TYPE ST_SortStationParam :
STRUCT
	lrGoodPosition 		: LREAL;
	tGoodTimer			: TIME;
	
	lrDirtPosition 		: LREAL;
	tDirtTimer			: TIME;
	
	lrDentPosition 		: LREAL;
	tDentTimer			: TIME;
	
	lrRejectPosition 	: LREAL;
	tRejectTimer		: TIME;
	
END_STRUCT
END_TYPE

(* stored: Version 1.1.0.1, ProductVersion 3.1.4024.9
   DUT ST_SortStationParam: Id {b958e278-eeda-4e1e-99ce-beb538959e53} *)
